// TIA Portal V20 export
TYPE "LER_typeVisionData"
// stored: Access Published
   STRUCT
      VisionOk : Bool;
      VisionNG : Bool;
      VisionComplete : Bool;
      GagueRnR_Type1OK : Bool;
      GagueRnR_Type1NG : Bool;
      GagueRnR_Type1Complete : Bool;
      GagueRnR_Type3OK : Bool;
      GagueRnR_Type3NG : Bool;
      GagueRnR_Type3Complete : Bool;
      VisionData : "LER_typeVisionResultData";
   END_STRUCT;
END_TYPE
